% RSLogix 500 project Project 3.RSS, saved by version 8.30.00.16 %
PROJECT "UNTITLED"    % processor: Bul.1763 MicroLogix 1100 Series B %

PROGRAM FILES
  LAD 2   10 rungs

DATA FILES
  O0 OUTPUT  4 elements
  I1 INPUT  6 elements
  S2 STATUS  66 elements
  B3 BINARY  1 elements
  T4 TIMER  1 elements
  C5 COUNTER  1 elements
  R6 CONTROL  1 elements
  N7 INTEGER  12 elements
  F8 FLOAT  1 elements
  ST9 STRING  7 elements

LADDER 2
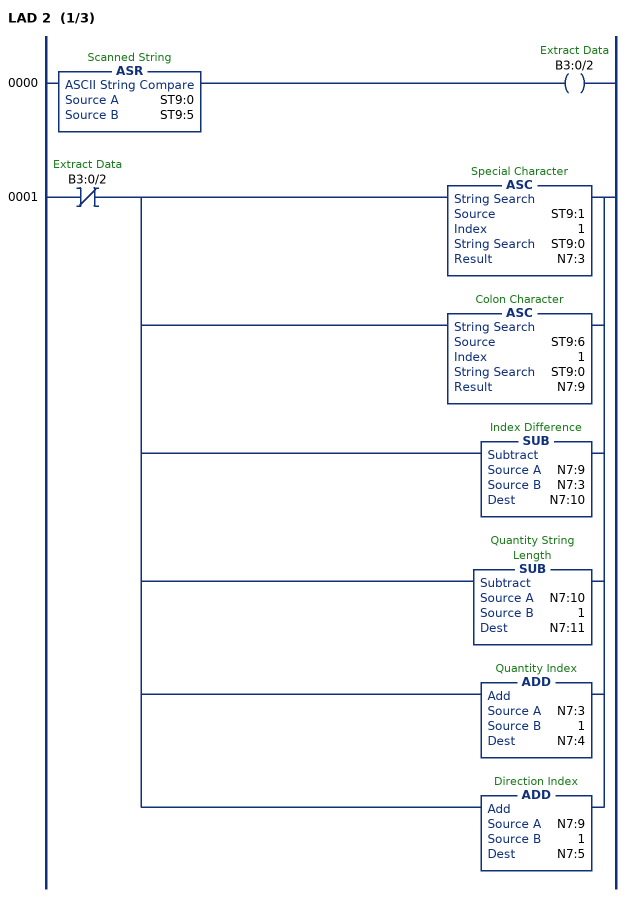
% Rung: 0 %
SOR ASR ST9:0 ST9:5 OTE B3:0/2 EOR
%   ST9:0  "Scanned String" %
%   ST9:5  "Empty String" %
%   B3:0/2  "Extract Data" %
% Rung: 1 %
SOR XIO B3:0/2 BST ASC ST9:1 1 ST9:0 N7:3 NXB ASC ST9:6 1 ST9:0 N7:9 NXB SUB N7:9 N7:3 N7:10 NXB SUB N7:10 1 N7:11 NXB ADD N7:3 1 N7:4 NXB ADD N7:9 1 N7:5 BND EOR
%   B3:0/2  "Extract Data" %
%   ST9:1  "Special Character" %
%   ST9:0  "Scanned String" %
%   N7:3  "Index of -" %
%   ST9:6  "Colon Character" %
%   N7:9  "Colon Index" %
%   N7:10  "Index Difference" %
%   N7:11  "Quantity String Length" %
%   N7:4  "Quantity Index" %
%   N7:5  "Direction Index" %

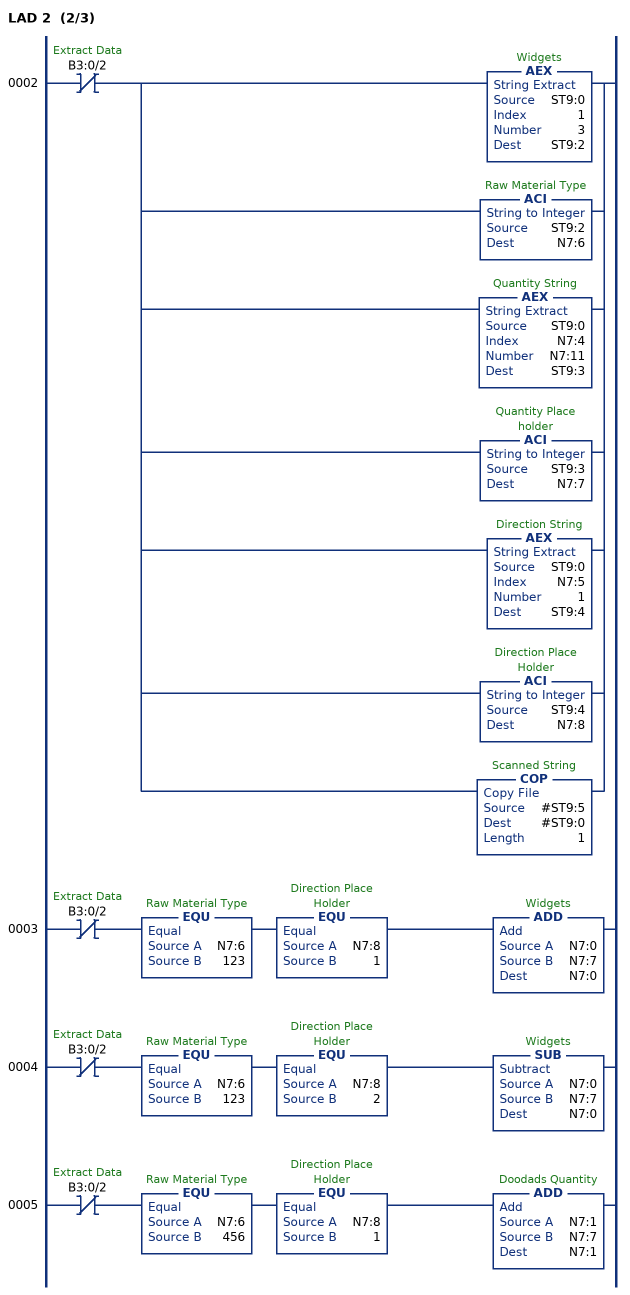
% Rung: 2 %
SOR XIO B3:0/2 BST AEX ST9:0 1 3 ST9:2 NXB ACI ST9:2 N7:6 NXB AEX ST9:0 N7:4 N7:11 ST9:3 NXB ACI ST9:3 N7:7 NXB AEX ST9:0 N7:5 1 ST9:4 NXB ACI ST9:4 N7:8 NXB COP #ST9:5 #ST9:0 1 BND EOR
%   B3:0/2  "Extract Data" %
%   ST9:0  "Scanned String" %
%   ST9:2  "Widgets" %
%   N7:6  "Raw Material Type" %
%   N7:4  "Quantity Index" %
%   N7:11  "Quantity String Length" %
%   ST9:3  "Quantity String" %
%   N7:7  "Quantity Place holder" %
%   N7:5  "Direction Index" %
%   ST9:4  "Direction String" %
%   N7:8  "Direction Place Holder" %
%   ST9:5  "Empty String" %
% Rung: 3 %
SOR XIO B3:0/2 EQU N7:6 123 EQU N7:8 1 ADD N7:0 N7:7 N7:0 EOR
%   B3:0/2  "Extract Data" %
%   N7:6  "Raw Material Type" %
%   N7:8  "Direction Place Holder" %
%   N7:0  "Widgets" %
%   N7:7  "Quantity Place holder" %
% Rung: 4 %
SOR XIO B3:0/2 EQU N7:6 123 EQU N7:8 2 SUB N7:0 N7:7 N7:0 EOR
%   B3:0/2  "Extract Data" %
%   N7:6  "Raw Material Type" %
%   N7:8  "Direction Place Holder" %
%   N7:0  "Widgets" %
%   N7:7  "Quantity Place holder" %
% Rung: 5 %
SOR XIO B3:0/2 EQU N7:6 456 EQU N7:8 1 ADD N7:1 N7:7 N7:1 EOR
%   B3:0/2  "Extract Data" %
%   N7:6  "Raw Material Type" %
%   N7:8  "Direction Place Holder" %
%   N7:1  "Doodads Quantity" %
%   N7:7  "Quantity Place holder" %

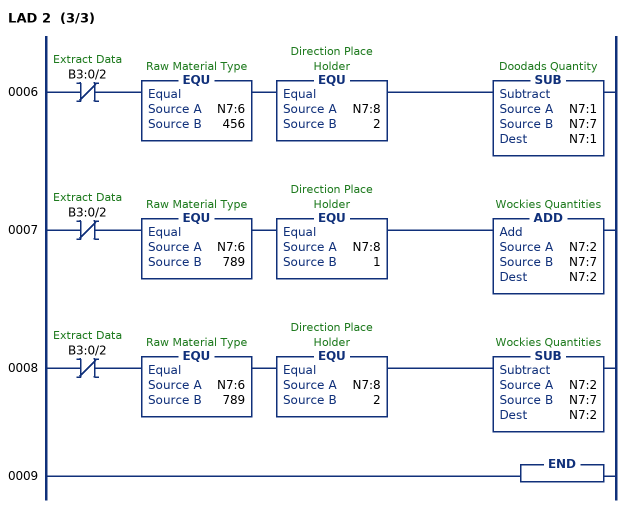
% Rung: 6 %
SOR XIO B3:0/2 EQU N7:6 456 EQU N7:8 2 SUB N7:1 N7:7 N7:1 EOR
%   B3:0/2  "Extract Data" %
%   N7:6  "Raw Material Type" %
%   N7:8  "Direction Place Holder" %
%   N7:1  "Doodads Quantity" %
%   N7:7  "Quantity Place holder" %
% Rung: 7 %
SOR XIO B3:0/2 EQU N7:6 789 EQU N7:8 1 ADD N7:2 N7:7 N7:2 EOR
%   B3:0/2  "Extract Data" %
%   N7:6  "Raw Material Type" %
%   N7:8  "Direction Place Holder" %
%   N7:2  "Wockies Quantities" %
%   N7:7  "Quantity Place holder" %
% Rung: 8 %
SOR XIO B3:0/2 EQU N7:6 789 EQU N7:8 2 SUB N7:2 N7:7 N7:2 EOR
%   B3:0/2  "Extract Data" %
%   N7:6  "Raw Material Type" %
%   N7:8  "Direction Place Holder" %
%   N7:2  "Wockies Quantities" %
%   N7:7  "Quantity Place holder" %
% Rung: 9 %
SOR END EOR

OTHER DOCUMENTED ADDRESSES
  B3:0/0  "Fire Once"
  B3:0/1  "Data Extracted"
  B3:0/3  "Move Data"
  B3:0/4  "Fire Once"
  B3:0/5  "Widgets Moved"
  B3:0/6  "Doodads Moved"
  B3:0/7  "Wockies Moved"
  B3:0/8  "Fire Once"
  B3:0/9  "FIre Once"
  B3:0/10  "Fire Once"
  B3:0/11  "Fire Once"
  B3:0/12  "Fire Once"
  B3:0/13  "Fire Once"

DATA TABLE (non-zero values as saved)
DATA ST9
% ST9:1 % "-"
% ST9:6 % ":"
